{attribute addProperty BoxType "EP1122-0001-0018"}
{attribute addProperty Id "A_0027_EP1258_0001_0016EP1258_BB8E9A1042052.5A_0028_EP1258_0001_0017EP1258_BB8E9A1042052.5A_0029_EP1258_0001_0018EP1258_BB8E9A1042052.5A_0030_EP1258_0001_0019EP1258_BB8E9A1042052.5A_0031_EP1258_0001_0020EP1258_BB8E9A1042052.5A_0032_EP1258_0002_0016EP1258_BB8E9A1042052.5A_0033_EP1258_0002_0017EP1258_BB8E9A1042052.5A_0034_EP1258_0002_0018EP1258_BB8E9A1042052.5A_0035_EP1258_0002_0019EP1258_BB8E9A1042052.5A_0036_EP1258_0002_0020EP1258_BB8E9A1042052.5A_0037_EP1312_0001_0016A_0037_EP1312_0001_0016_91E425AA594268719477478.75"}
{attribute addProperty CRC "3236180118"}
{attribute addProperty SizeInBites "10142"}
{attribute addProperty SizeInBytes "68719478003.75"}
TYPE A_0026_EP1122_0001_0018_C0E43096 EXTENDS EP1122_179A0949 :
STRUCT
	{attribute addProperty Name "A_0027_EP1258_0001_0016"}
	A_0027_EP1258_0001_0016 : EP1258_BB8E9A10;
	{attribute addProperty Name "A_0028_EP1258_0001_0017"}
	A_0028_EP1258_0001_0017 : EP1258_BB8E9A10;
	{attribute addProperty Name "A_0029_EP1258_0001_0018"}
	A_0029_EP1258_0001_0018 : EP1258_BB8E9A10;
	{attribute addProperty Name "A_0030_EP1258_0001_0019"}
	A_0030_EP1258_0001_0019 : EP1258_BB8E9A10;
	{attribute addProperty Name "A_0031_EP1258_0001_0020"}
	A_0031_EP1258_0001_0020 : EP1258_BB8E9A10;
	{attribute addProperty Name "A_0032_EP1258_0002_0016"}
	A_0032_EP1258_0002_0016 : EP1258_BB8E9A10;
	{attribute addProperty Name "A_0033_EP1258_0002_0017"}
	A_0033_EP1258_0002_0017 : EP1258_BB8E9A10;
	{attribute addProperty Name "A_0034_EP1258_0002_0018"}
	A_0034_EP1258_0002_0018 : EP1258_BB8E9A10;
	{attribute addProperty Name "A_0035_EP1258_0002_0019"}
	A_0035_EP1258_0002_0019 : EP1258_BB8E9A10;
	{attribute addProperty Name "A_0036_EP1258_0002_0020"}
	A_0036_EP1258_0002_0020 : EP1258_BB8E9A10;
	{attribute addProperty Name "A_0037_EP1312_0001_0016"}
	A_0037_EP1312_0001_0016 : A_0037_EP1312_0001_0016_91E425AA;
END_STRUCT
END_TYPE

(* stored: Version 1.2.0.0, ProductVersion 3.1.4024.9
   DUT A_0026_EP1122_0001_0018_C0E43096: Id {2cc02de4-1a21-41a0-9ec0-d4ed5d166e02} *)
